Staubli VAL3: init.pgx

public program init()
  local bool ok
  local string path
  local num idx
begin
  // set module index
  path=libPath()
  path=right(path,1)
  path=toNum(path,moduleIndex,ok)
  if !ok
    moduleIndex=0
  endIf
  name="IMM"+toString("1.0",moduleIndex)
  IMM_IO_PTH="2:IO/1:"+name
  nCaseBtRobOff=1
  bState=false
  pointer=0
  for idx=0 to size(timings)-1
    timings[idx]=0
  endFor

end
